TYPE P_Axis_Rx :
STRUCT
	STATUS_WORD:UINT;
	POSITION_VALUE:DINT;
END_STRUCT
END_TYPE

(* stored: Version 1.1.0.1, ProductVersion 3.1.4024.12
   DUT P_Axis_Rx: Id {5fe60f1f-614e-427c-8128-0a8b238093ee} *)
